INTERFACE I_Observer

METHOD Update
VAR_INPUT	
	fValue			: LREAL;
END_VAR
END_METHOD

END_INTERFACE

(* stored: Version 1.1.0.1, ProductVersion 3.1.4022.7
   Itf I_Observer: Id {c58171d1-03b0-44cb-9810-3cafe2601289}
   Method Update: Id {addc419a-1b9f-4b31-943e-d5346d184248} *)
